INTERFACE I_VFD

METHOD Jog : BOOL
VAR_INPUT
    JogFW : BOOL := FALSE;
    JogBW : BOOL := FALSE;
END_VAR
END_METHOD

METHOD Stop : BOOL
VAR_INPUT
END_VAR
END_METHOD

END_INTERFACE

(* stored: Version 1.1.0.1
   Itf I_VFD: Id {d5046df4-1d79-44a2-92aa-463fd5a4ba92}
   Method Jog: Id {a9ea47fc-b360-443e-8b19-e74f56e72cfd}
   Method Stop: Id {092b1b8a-9c2e-4743-89cc-51249266c685} *)
